TYPE LimitSwitches :
(
	POSITIVE_LIMIT_SWITCH := 0,
	NEGATIVE_LIMIT_SWITCH := 1
);
END_TYPE

(* stored: Version 1.1.0.1, ProductVersion 3.1.4019.2
   DUT LimitSwitches: Id {c113c1ce-c5cb-4e01-a0af-afd5773ffb19} *)
